{attribute 'qualified_only'}
VAR_GLOBAL
	// 儲列使用計數器
	evenNumber		: UDINT;
	
	DoneNumber 		: UDINT;

	messageList : ARRAY[0..15] OF MsgStruct;
	
// SQL 執行命令型
_fb_PLCDBCmdEvt : FB_PLCDBCmdEvt(sNetID:= '', tTimeout:= T#5S );

	systime         : FB_LocalSystemTime;
	currentTime     : DT;
END_VAR

(* stored: Version 1.1.0.1, ProductVersion 3.1.4026.13
   GVL MsgBuff: Id {b0d33a80-77e8-4b5a-8915-a3316682a589} *)
